// TIA Portal V19 export
TYPE "udt_WeldReg_Pers"
   STRUCT
      CoilThreadingDone : Bool;
      WeldMeasInpID : UInt;
      WelderRegID : DInt;
      WelderReg : Array[1.."WELDER_ITEMS_QTY"] of "udt_WeldReg_Item";
      Par : Struct
         TP_On_InsideHole : Bool;
         TP_OffsetFromCut : LReal;
      END_STRUCT;
   END_STRUCT;
END_TYPE
